{attribute 'qualified_only'}
VAR_GLOBAL
	stValveOutWinch : ST_ValveOutputs;
	stValveOutCyl : ST_ValveOutputs; 
END_VAR

(* stored: Version 1.1.0.1, ProductVersion 3.1.4024.12
   GVL G_OutputList: Id {3e7d87a4-3f87-4f4e-83da-69e1364ee6d4} *)
